{attribute 'linkalways'} 
{attribute 'no_explicit_call' := 'This FB is a CLASS and must be accessed using methods or properties'}
{attribute 'enable_dynamic_creation'}
FUNCTION_BLOCK JsonDeserializerNullNode EXTENDS Disposable IMPLEMENTS I_Deserializer
VAR
	parent : I_JsonDeserializer;
END_VAR

METHOD PUBLIC Clone : I_Deserializer
VAR
	pClone : POINTER TO JsonDeserializerNullNode;
END_VAR
pClone := __NEW(JsonDeserializerNullNode(ParentJsonDeserializer := parent));
Clone := pClone^;
END_METHOD

METHOD PROTECTED CreateNullEnumerator : I_DeserializerForwardEnumerator
VAR_INPUT
END_VAR
VAR
	pForwardEnumerator : POINTER TO JsonDeserializerNullForwardEnumerator;
END_VAR
pForwardEnumerator := __NEW(JsonDeserializerNullForwardEnumerator(ParentJsonDeserializer := parent, ParentNullDeserializer := THIS^));
CreateNullEnumerator := pForwardEnumerator^;
END_METHOD

METHOD FB_init : BOOL
VAR_INPUT
	bInitRetains : BOOL; // if TRUE, the retain variables are initialized (warm start / cold start)
	bInCopyCode : BOOL;  // if TRUE, the instance afterwards gets moved into the copy code (online change)
	ParentJsonDeserializer : I_JsonDeserializer;
END_VAR
THIS^.parent := ParentJsonDeserializer;
END_METHOD

METHOD GetArray : I_Deserializer
VAR_INPUT
END_VAR
GetArray := this^;
END_METHOD

METHOD GetArrayElementEnumerator : I_DeserializerForwardEnumerator
VAR_INPUT
END_VAR
GetArrayElementEnumerator := CreateNullEnumerator();
END_METHOD

METHOD GetElementByIndex : I_Deserializer
VAR_INPUT
	Index : UDINT;
END_VAR
GetElementByIndex := this^;
END_METHOD

METHOD GetKey : I_Deserializer
VAR_INPUT
	Key : T_MAXSTRING;
END_VAR
GetKey := this^;
END_METHOD

METHOD GetKeyArray : I_Deserializer
VAR_INPUT
	Key : T_MAXSTRING;
END_VAR
GetKeyArray := this^;
END_METHOD

METHOD GetObjectKeyEnumerator : I_DeserializerForwardEnumerator
VAR_INPUT
END_VAR
GetObjectKeyEnumerator := CreateNullEnumerator();
END_METHOD

METHOD TryGetBase64 : BOOL
VAR_INPUT
	pBytes : POINTER TO BYTE;
	nBytes : DINT;
END_VAR
END_METHOD

METHOD TryGetBool : BOOL
VAR_INPUT
	Destination : REFERENCE TO BOOL;
END_VAR
END_METHOD

METHOD TryGetByte : BOOL
VAR_INPUT
	Destination : REFERENCE TO BYTE;
END_VAR
END_METHOD

METHOD TryGetDateTime : BOOL
VAR_INPUT
	Destination : REFERENCE TO DATE_AND_TIME;
END_VAR
END_METHOD

METHOD TryGetDcTime : BOOL
VAR_INPUT
	Destination : REFERENCE TO DCTIME;
END_VAR
END_METHOD

METHOD TryGetDint : BOOL
VAR_INPUT
	Destination : REFERENCE TO DINT;
END_VAR
END_METHOD

METHOD TryGetDword : BOOL
VAR_INPUT
	Destination : REFERENCE TO DWORD;
END_VAR
END_METHOD

METHOD TryGetFileTime : BOOL
VAR_INPUT
	Destination : REFERENCE TO FILETIME;
END_VAR
END_METHOD

METHOD TryGetHexAsBytes : BOOL
VAR_INPUT
	pBytes : POINTER TO BYTE;
	nBytes : DINT;
END_VAR
END_METHOD

METHOD TryGetInt : BOOL
VAR_INPUT
	Destination : REFERENCE TO INT;
END_VAR
END_METHOD

METHOD TryGetKeyBase64 : BOOL
VAR_INPUT
	Key : T_MAXSTRING;
	pBytes : POINTER TO BYTE;
	nBytes : DINT;
END_VAR
END_METHOD

METHOD TryGetKeyBool : BOOL
VAR_INPUT
	Key : T_MAXSTRING;
	Destination : REFERENCE TO BOOL;
END_VAR
END_METHOD

METHOD TryGetKeyByte : BOOL
VAR_INPUT
	Key : T_MAXSTRING;
	Destination : REFERENCE TO BYTE;
END_VAR
END_METHOD

METHOD TryGetKeyDateTime : BOOL
VAR_INPUT
	Key : T_MAXSTRING;
	Destination : REFERENCE TO DATE_AND_TIME;
END_VAR
END_METHOD

METHOD TryGetKeyDcTime : BOOL
VAR_INPUT
	Key : T_MAXSTRING;
	Destination : REFERENCE TO DCTIME;
END_VAR
END_METHOD

METHOD TryGetKeyDint : BOOL
VAR_INPUT
	Key : T_MAXSTRING;
	Destination : REFERENCE TO DINT;
END_VAR
END_METHOD

METHOD TryGetKeyDword : BOOL
VAR_INPUT
	Key : T_MAXSTRING;
	Destination : REFERENCE TO DWORD;
END_VAR
END_METHOD

METHOD TryGetKeyFileTime : BOOL
VAR_INPUT
	Key : T_MAXSTRING;
	Destination : REFERENCE TO FILETIME;
END_VAR
END_METHOD

METHOD TryGetKeyHexAsBytes : BOOL
VAR_INPUT
	Key : T_MAXSTRING;
	pBytes : POINTER TO BYTE;
	nBytes : DINT;
END_VAR
END_METHOD

METHOD TryGetKeyInt : BOOL
VAR_INPUT
	Key : T_MAXSTRING;
	Destination : REFERENCE TO INT;
END_VAR
END_METHOD

METHOD TryGetKeyLint : BOOL
VAR_INPUT
	Key : T_MAXSTRING;
	Destination : REFERENCE TO LINT;
END_VAR
END_METHOD

METHOD TryGetKeyLreal : BOOL
VAR_INPUT
	Key : T_MAXSTRING;
	Destination : REFERENCE TO LREAL;
END_VAR
END_METHOD

METHOD TryGetKeyLtime : BOOL
VAR_INPUT
	Key : T_MAXSTRING;
	Destination : REFERENCE TO LTIME;
END_VAR
END_METHOD

METHOD TryGetKeyLword : BOOL
VAR_INPUT
	Key : T_MAXSTRING;
	Destination : REFERENCE TO LWORD;
END_VAR
END_METHOD

METHOD TryGetKeyObject : BOOL
VAR_INPUT
	Key : T_MAXSTRING;
	Object : I_Deserializable;
END_VAR
END_METHOD

METHOD TryGetKeyReal : BOOL
VAR_INPUT
	Key : T_MAXSTRING;
	Destination : REFERENCE TO REAL;
END_VAR
END_METHOD

METHOD TryGetKeySint : BOOL
VAR_INPUT
	Key : T_MAXSTRING;
	Destination : REFERENCE TO SINT;
END_VAR
END_METHOD

METHOD TryGetKeyString : BOOL
VAR_INPUT
	Key : T_MAXSTRING;
	Destination : REFERENCE TO STRING;
END_VAR
END_METHOD

METHOD TryGetKeyTime : BOOL
VAR_INPUT
	Key : T_MAXSTRING;
	Destination : REFERENCE TO TIME;
END_VAR
END_METHOD

METHOD TryGetKeyTod : BOOL
VAR_INPUT
	Key : T_MAXSTRING;
	Destination : REFERENCE TO TOD;
END_VAR
END_METHOD

METHOD TryGetKeyUdint : BOOL
VAR_INPUT
	Key : T_MAXSTRING;
	Destination : REFERENCE TO UDINT;
END_VAR
END_METHOD

METHOD TryGetKeyUint : BOOL
VAR_INPUT
	Key : T_MAXSTRING;
	Destination : REFERENCE TO UINT;
END_VAR
END_METHOD

METHOD TryGetKeyUlint : BOOL
VAR_INPUT
	Key : T_MAXSTRING;
	Destination : REFERENCE TO ULINT;
END_VAR
END_METHOD

METHOD TryGetKeyUsint : BOOL
VAR_INPUT
	Key : T_MAXSTRING;
	Destination : REFERENCE TO USINT;
END_VAR
END_METHOD

METHOD TryGetKeyWord : BOOL
VAR_INPUT
	Key : T_MAXSTRING;
	Destination : REFERENCE TO WORD;
END_VAR
END_METHOD

METHOD TryGetLint : BOOL
VAR_INPUT
	Destination : REFERENCE TO LINT;
END_VAR
END_METHOD

METHOD TryGetLreal : BOOL
VAR_INPUT
	Destination : REFERENCE TO LREAL;
END_VAR
END_METHOD

METHOD TryGetLtime : BOOL
VAR_INPUT
	Destination : REFERENCE TO LTIME;
END_VAR
END_METHOD

METHOD TryGetLword : BOOL
VAR_INPUT
	Destination : REFERENCE TO LWORD;
END_VAR
END_METHOD

METHOD TryGetName : BOOL
VAR_INPUT
	Destination : REFERENCE TO STRING;
END_VAR
END_METHOD

METHOD TryGetObject : BOOL
VAR_INPUT
	Object : I_Deserializable;
END_VAR
END_METHOD

METHOD TryGetReal : BOOL
VAR_INPUT
	Destination : REFERENCE TO REAL;
END_VAR
END_METHOD

METHOD TryGetSint : BOOL
VAR_INPUT
	Destination : REFERENCE TO SINT;
END_VAR
END_METHOD

METHOD TryGetString : BOOL
VAR_INPUT
	Destination : REFERENCE TO STRING;
END_VAR
END_METHOD

METHOD TryGetTime : BOOL
VAR_INPUT
	Destination : REFERENCE TO TIME;
END_VAR
END_METHOD

METHOD TryGetTod : BOOL
VAR_INPUT
	Destination : REFERENCE TO TOD;
END_VAR
END_METHOD

METHOD TryGetUdint : BOOL
VAR_INPUT
	Destination : REFERENCE TO UDINT;
END_VAR
END_METHOD

METHOD TryGetUint : BOOL
VAR_INPUT
	Destination : REFERENCE TO UINT;
END_VAR
END_METHOD

METHOD TryGetUlint : BOOL
VAR_INPUT
	Destination : REFERENCE TO ULINT;
END_VAR
END_METHOD

METHOD TryGetUsint : BOOL
VAR_INPUT
	Destination : REFERENCE TO USINT;
END_VAR
END_METHOD

METHOD TryGetWord : BOOL
VAR_INPUT
	Destination : REFERENCE TO WORD;
END_VAR
END_METHOD

END_FUNCTION_BLOCK

(* stored: Version 1.1.0.1, ProductVersion 3.1.4024.12
   POU JsonDeserializerNullNode: Id {6b115126-7669-4eaa-a7e3-ffc35f98e823}, SpecialFunc None
   Folder Constructor: Id {61e75f43-1ee7-40b9-bb04-a038519b40d9}
   Folder Protected: Id {7a59f1c0-5241-4e62-94fc-3dbb0a948e73}
   Method Clone: Id {3f922643-7671-4c7a-a549-0c960b9d0b10}
   Method CreateNullEnumerator: Id {cb2fe48b-2345-4050-8de9-290676488da6}
   Method FB_init: Id {1e7296e9-f185-4ade-9915-6f5f29e97c6c}
   Method GetArray: Id {f493d27e-bbbd-46ae-af30-5daf1dfbd856}
   Method GetArrayElementEnumerator: Id {a88ad026-4ec7-4218-9ece-bf13af031698}
   Method GetElementByIndex: Id {4678a701-0ece-47f5-87d0-50c6ccbaaabd}
   Method GetKey: Id {09b29dfb-1cd9-4ffc-8847-0eb0c4907f31}
   Method GetKeyArray: Id {13143476-2862-4c41-a794-22b9488d0f09}
   Method GetObjectKeyEnumerator: Id {a7b69884-3b2b-4b72-863d-2e0e1feccd98}
   Method TryGetBase64: Id {f75b94cc-09a1-46d1-96bc-828dc273232b}
   Method TryGetBool: Id {1482a02b-44b1-4d00-83d0-bfcbd02aa9e5}
   Method TryGetByte: Id {11cb8760-de5a-4d4a-abb4-721cead140d7}
   Method TryGetDateTime: Id {659f2c53-3753-422e-9477-31d422b9487e}
   Method TryGetDcTime: Id {19769951-7c91-4379-84fd-7686a89ea8e8}
   Method TryGetDint: Id {8aa00f02-1abe-4580-99ff-357eec4747da}
   Method TryGetDword: Id {fe7aefa0-2ba8-4edf-b2a1-24f237ca79dc}
   Method TryGetFileTime: Id {37fea43a-0d3d-41c5-bca3-a8674c31e111}
   Method TryGetHexAsBytes: Id {ff79c0d4-f18a-4054-ba59-43211cefaef3}
   Method TryGetInt: Id {c0ac5635-3443-487e-8b70-ca8a8e83ad64}
   Method TryGetKeyBase64: Id {d609f69b-8d67-4fed-a81d-2159cdd224d4}
   Method TryGetKeyBool: Id {3949d21f-ee79-496e-b495-9d95e7fedfad}
   Method TryGetKeyByte: Id {f6504235-e1c1-4387-bdbc-9b85ba59e4d1}
   Method TryGetKeyDateTime: Id {8101862d-5f18-441e-ad08-b13eab9da495}
   Method TryGetKeyDcTime: Id {27f56608-dbac-438d-a941-c37cc857326e}
   Method TryGetKeyDint: Id {680ad871-fb84-4e71-9045-204b8b36c8dd}
   Method TryGetKeyDword: Id {5e9754ab-bf9b-4141-bfc7-dde1a7fa1e53}
   Method TryGetKeyFileTime: Id {01285bcb-0898-4dbf-beab-41ec85c9c99c}
   Method TryGetKeyHexAsBytes: Id {a4ff13b2-bfa9-4641-9ba7-f0ec9882b9ad}
   Method TryGetKeyInt: Id {ead7d035-34f5-409c-a51c-6e193dcb8920}
   Method TryGetKeyLint: Id {be3b394b-9380-4dd9-9a90-ae11e7807234}
   Method TryGetKeyLreal: Id {177564d9-01c8-4f12-b3ad-c87503590719}
   Method TryGetKeyLtime: Id {d22a41f7-9170-4d5b-aa93-439e3d810188}
   Method TryGetKeyLword: Id {fa4c3522-3bfd-41e7-9ba8-aedee884521d}
   Method TryGetKeyObject: Id {695f142e-e075-4776-8893-232de584ac13}
   Method TryGetKeyReal: Id {3a66a959-2786-4929-b7a9-0744eb355910}
   Method TryGetKeySint: Id {fe7a5584-ccdc-41a2-811b-6bef1a753e08}
   Method TryGetKeyString: Id {5d897420-9d9f-4549-910c-633714336499}
   Method TryGetKeyTime: Id {daca10e0-ba1f-4329-ba30-e0fa923de2c7}
   Method TryGetKeyTod: Id {078b2bc5-7fb6-470a-992c-f362fd2eed22}
   Method TryGetKeyUdint: Id {c0fce314-bb1f-44a3-8a2c-f7234aa13a5c}
   Method TryGetKeyUint: Id {df0356db-c14b-43ba-b6dd-d54246c11a5c}
   Method TryGetKeyUlint: Id {d4e69df0-8b22-439e-90db-e0bd326bbc68}
   Method TryGetKeyUsint: Id {d9a54d8d-cf3e-4d8e-9492-2539fbcc1e0b}
   Method TryGetKeyWord: Id {49c7544e-be1a-42a3-b879-6c2651e791f2}
   Method TryGetLint: Id {a2e62477-ec1e-4c8e-8605-b260650cec0e}
   Method TryGetLreal: Id {d3c4d08f-578b-4d47-8b61-660aee4b562b}
   Method TryGetLtime: Id {d9901346-0e98-4947-a628-664e46cb87be}
   Method TryGetLword: Id {48a98534-9d79-425c-abf7-b55251dede15}
   Method TryGetName: Id {10517808-4411-487f-8a6b-f34a550ffb2d}
   Method TryGetObject: Id {875341c4-f0f4-4402-8e37-703bc59a9101}
   Method TryGetReal: Id {15967a65-c0a8-4588-b15a-7ce8296db26e}
   Method TryGetSint: Id {00611a3c-0448-48c0-a2d7-87db39f4ba5d}
   Method TryGetString: Id {953f735b-7fb0-4fd8-8e11-7a9c8f4ddf7b}
   Method TryGetTime: Id {057bac58-daa6-4023-91ac-dd7165e53c8f}
   Method TryGetTod: Id {917ec393-ae8d-490a-a5d4-2f12beab5406}
   Method TryGetUdint: Id {c16e53e7-ff8f-46b7-90dd-cf5e00432c65}
   Method TryGetUint: Id {dabc74d4-3664-4d7a-ac1d-a1dea7bc5e0e}
   Method TryGetUlint: Id {c090dd5c-eab4-49e5-ac25-7d01148e5c33}
   Method TryGetUsint: Id {1f92fef4-23a9-43fc-aa7c-cbb835cf680e}
   Method TryGetWord: Id {21f5aa0b-e03d-4303-96fe-efdd965c95cf} *)
